{attribute 'qualified_only'}
VAR_GLOBAL
	DataFromHmi	: _DATA_FROM_HMI;
	DataToHmi	: _DATA_TO_HMI;
END_VAR

(* stored: Version 1.1.0.1, ProductVersion 3.1.4024.16
   GVL GVL: Id {208ffac8-2a3f-4c68-b764-9237f82d26ca} *)
